(* CoDeSys 2.3.9.41 project: Coffee.pro *)
(* Libraries: Standard.lib 4.10.05 11:14:46, IecSfc.lib 13.4.06 15:51:28, SYSLIBCALLBACK.LIB 26.9.08 16:43:52 *)

(* Global variable list: Global_Variables *)
VAR_GLOBAL
 	(*------------входы--------------*)

	(*-----------кнопки-------------*)
	start:BOOL; (*пуск*)
	emergency_stop:BOOL; (*аварийная остановка*)
	stop: BOOL; (*плавное завершение*)
	plus: BOOL; (*количество порций +1*)
	minus:BOOL; (*количество порций -1*)

	(*-----------датчики------------*)
	upper_temperature:BOOL; (*верхняя температура*)
	lower_temperature:BOOL; (*нижняя температура*)
	working_temperature:BOOL; (*рабочая температура*)
	water_level_sensor:BOOL; (*датчик уровня воды*)


	(*-----------выходы------------*)

	(*-------Устройства / Лампы--------*)
	(*---------нагреватель-------------*)
	turn_on_the_heater:BOOL; (*включить нагреватель*)
	(*---------клапаны-----------*)
	open_the_valve_1:BOOL; (*открыть клапан 1*)
	open_the_valve_2:BOOL; (*открыть клапан 2*)

	(*--------Режимы / Лампы----------*)
	(*--------режим работы-------------*)
	water_supply:BOOL; (*подача воды*)
	steam_release:BOOL; (*выпуск пара*)
	heating_boiling:BOOL; (*нагревание/кипячение*)

	(*---------Состояния / Лампы---------*)
	(*----------система-----------*)
	system_is_on:BOOL; (*система включена*)
	smooth_ending:BOOL; (*плавное завершение*)
	emergency_stopp:BOOL; (*аварийная остановка*)
	(*--------нагреватель/температура---------*)
	upper_temperaturee:BOOL; (*верхняя температура*)
	lower_temperaturee:BOOL; (*нижняя температура*)
	working_temperaturee:BOOL; (*рабочая температура*)
	the_heater_is_faulty:BOOL; (*нагреватель неисправен*)
	(*-------псевдодатчики-------*)
	level_0_in_the_tank:BOOL;(*уровень 0 в емкости*)
	level_1_in_the_tank:BOOL; (*уровень 1 в емкости*)
	steam_pressure_in_the_tank:BOOL; (*пар/давление в емкости*)
	(*------дисплей-------*)
	first_rank:BOOL; (*первый разряд числа*)
	second_rank:BOOL; (*второй разряд числа*)
	third_rank:BOOL; (*третий разряд числа*)
	(*--------уровень--------*)
	water_level_is_normal:BOOL; (*уровень воды в норме*)

	(*----таймеры----*)
	DropTimer: TON := (PT := T#3s); (*таймер выпуска пара через клапаны*)
	timer_for_second_valve: TON:= (PT := T#3s);

END_VAR

(* POU PLC_PRG, ST *)
PROGRAM PLC_PRG
VAR
	pouring_water:BOOL;
	_level_0_in_the_tank:BOOL; (*уровень 0 в емкости*)
	_level_1_in_the_tank:BOOL;  (*уровень 1 в емкости*)
	_open_the_valve_1:BOOL; (*открыть клапан 1*)
	_open_the_valve_2:BOOL; (*открыть клапан 2*)

END_VAR
(*Уровень 0*)
IF NOT _level_0_in_the_tank AND _open_the_valve_1 AND water_level_sensor THEN
	level_0_in_the_tank := TRUE;

ELSIF _level_0_in_the_tank AND _open_the_valve_2 AND DropTimer.Q THEN
	level_0_in_the_tank := FALSE;
END_IF;


(*уровень 1*)

IF NOT _level_1_in_the_tank AND _open_the_valve_1 AND timer_for_second_valve.Q THEN
	level_1_in_the_tank := TRUE;

ELSIF _level_1_in_the_tank AND _open_the_valve_2 THEN
	level_0_in_the_tank := FALSE;
END_IF;
END_PROGRAM

(* Visualisation Coffee
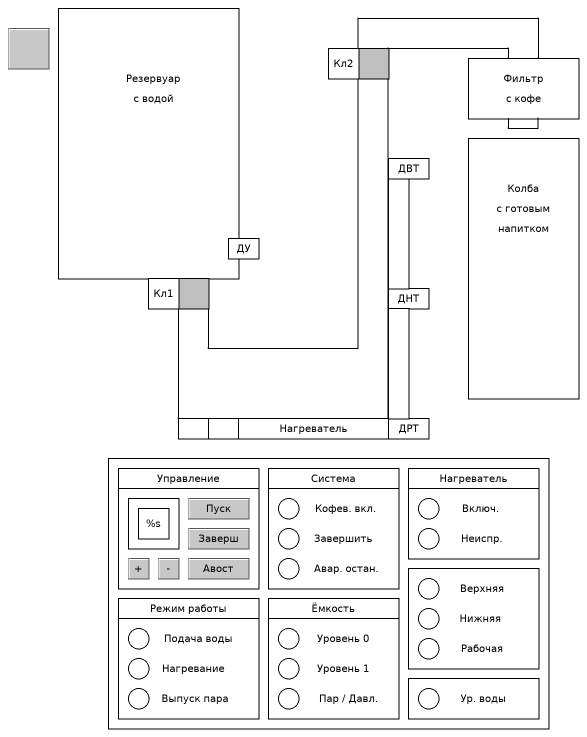
rectangle at (160,300)-(191,331): text "Кл1"
rectangle at (250,440)-(401,461): text "Нагреватель"
rectangle at (400,440)-(441,461): text "ДРТ"
rectangle at (400,310)-(441,331): text "ДНТ"
rectangle at (400,180)-(441,201): text "ДВТ"
rectangle at (240,260)-(271,281): text "ДУ"
rectangle at (130,490)-(271,511): text "Управление"
rectangle at (280,490)-(411,511): text "Система"
rectangle at (420,490)-(551,511): text "Нагреватель"
rectangle at (280,510)-(411,611): toggles свсв
rectangle at (280,620)-(411,641): text "Ёмкость"
rectangle at (150,530)-(181,561): text "%s"
button at (140,580)-(161,601): text "+"
button at (170,580)-(191,601): text "-"
button at (200,520)-(261,541): text "Пуск"
button at (200,550)-(261,571): text "Заверш"
button at (200,580)-(261,601): text "Авост"
rectangle at (130,620)-(271,641): text "Режим работы"
rectangle at (320,650)-(391,671): text "Уровень 0"
rectangle at (320,710)-(401,731): text "Пар / Давл."
rectangle at (320,680)-(391,701): text "Уровень 1"
rectangle at (320,580)-(391,601): text "Авар. остан."
rectangle at (320,550)-(391,571): text "Завершить"
rectangle at (320,520)-(401,541): text "Кофев. вкл."
rectangle at (460,660)-(531,681): text "Рабочая"
rectangle at (460,630)-(531,651): text "Нижняя"
rectangle at (460,600)-(531,621): text "Верхняя"
rectangle at (460,550)-(531,571): text "Неиспр."
rectangle at (460,520)-(531,541): text "Включ."
rectangle at (460,710)-(531,731): text "Ур. воды"
rectangle at (170,650)-(251,671): text "Подача воды"
rectangle at (170,710)-(241,731): text "Выпуск пара"
rectangle at (170,680)-(241,701): text "Нагревание"
rectangle at (340,70)-(371,101): text "Кл2"
rectangle at (130,110)-(201,131): text "с водой"
rectangle at (130,90)-(201,111): text "Резервуар"
rectangle at (500,90)-(571,111): text "Фильтр"
rectangle at (500,110)-(571,131): text "с кофе"
rectangle at (500,240)-(571,261): text "напитком"
rectangle at (500,220)-(571,241): text "с готовым"
rectangle at (500,200)-(571,221): text "Колба"
36 more shapes without text or variables
*)
